# EPICS substitutions: siteApps/EtherCat/m-epics-ecat2db/db/ecat2el2502.substitutions
file ecat2slave.template
{
	pattern {DEVICENAME}
		{EL2502}
}

file ecat2el250x.template
{
	pattern {CH_ID, PDO_IDX}
		{$(MOD_ID)-DO1, 0}
		{$(MOD_ID)-DO2, 1}
}
